{attribute addProperty BoxType "EL3681-0000-0018"}
{attribute addProperty Id "SAI_InputsAT %I*SAI_Inputs_6167285A4860SAI_RangeAT %I*SAI_Range_DF9848341620SAI_Range_1AT %Q*SAI_Range_80D0ED7D1620WcStateAT %I*WcState_F855686C1620InfoDataAT %I*InfoData_BC63D37F80100"}
{attribute addProperty CRC "649520245"}
{attribute addProperty SizeInBites "176"}
{attribute addProperty SizeInBytes "22"}
TYPE EL3681_7DAD71F7 :
STRUCT
	{attribute addProperty Name "SAI_Inputs"}
	SAI_Inputs : SAI_Inputs_6167285A;
	{attribute addProperty Name "SAI_Range"}
	SAI_Range : SAI_Range_DF984834;
	{attribute addProperty Name "SAI_Range_1"}
	SAI_Range_1 : SAI_Range_80D0ED7D;
	{attribute addProperty Name "WcState"}
	WcState : WcState_F855686C;
	{attribute addProperty Name "InfoData"}
	InfoData : InfoData_BC63D37F;
END_STRUCT
END_TYPE

(* stored: Version 1.2.0.0, ProductVersion 3.1.4024.9
   DUT EL3681_7DAD71F7: Id {4fc4639a-4ff1-4459-989d-94a6c70118bb} *)
